   A_21_A700Z1.CmdFaultReset := FALSE;
   A_21_A700Z1.InLocal := FALSE;
   A_21_A700Z1.spare0305 := FALSE;
   A_21_A700Z1.InReport := FALSE;
   A_21_A700Z1.OutTimeoutTime := FALSE;
   A_21_A700Z1.InHWStop := FALSE;
   A_21_A700Z1.InDPFault := FALSE;
   A_21_A700Z1.OutPreAlarmTrue := FALSE;
   A_21_A700Z1.OutPreAlarmFalse := FALSE;
   A_21_A700Z1.OutFlagPos := FALSE;
   A_21_A700Z1.OutFlagNeg := FALSE;
   A_21_A700Z1.OutpFaultReset := FALSE;
   A_21_A700Z1.OutTrue := FALSE;
   A_21_A700Z1.StFalse := FALSE;
   A_21_A700Z1.StCtoTrue := FALSE;
   A_21_A700Z1.StTrue := FALSE;
   A_21_A700Z1.StCtoFalse := FALSE;
   A_21_A700Z1.StFault := FALSE;
   A_21_A700Z1.OutAlarmNrLog := 0;
   A_21_A700Z1.Par.ParObjectNo := 533;
   A_21_A700Z1.Par.ParMsgType := 7147;
   A_21_A700Z1.Par.ParHornCode := 2;
   A_21_A700Z1.Par.ParLogOff := FALSE;
   A_21_A700Z1.Par.spare0401 := FALSE;
   A_21_A700Z1.Par.Par2WorkingCond := FALSE;
   A_21_A700Z1.Par.ParFaultRetry := FALSE;
   A_21_A700Z1.Par.ParBinLevel := FALSE;
   A_21_A700Z1.Par.ParDelayChange := 0;
   A_21_A700Z1.Par.ParDelayTrue := 10;
   A_21_A700Z1.Par.ParDelayFalse := 0;
   A_21_A700Z1.Par.ParTimeoutTrue := 0;
   A_21_A700Z1.Par.ParTimeoutFalse := 0;
   A_21_A700Z1.Par.OutMonTime := 0;
   A_21_A700Z1.Par.OutTransitionTime := 0;
   A_21_A700Z1.Par.OutMonTrue := FALSE;
   A_21_A700Z1.Par.OutMonFalse := FALSE;
   A_21_A700Z1.Par.OutFlagFaultDev := FALSE;
   A_21_A700Z1.Par.OutDelayTime := 0;
   A_21_A800Z1.StCode := 0;
   A_21_A800Z1.InMonTrue := FALSE;
   A_21_A800Z1.InMonFalse := FALSE;
   A_21_A800Z1.InPreAlarmTrue := FALSE;
   A_21_A800Z1.InPreAlarmFalse := FALSE;
   A_21_A800Z1.InStopTrueTime := FALSE;
   A_21_A800Z1.InStopFalseTime := FALSE;
   A_21_A800Z1.InpTrue := FALSE;
   A_21_A800Z1.InpFaultDev := FALSE;
   A_21_A800Z1.CmdRstTrueTime := FALSE;
   A_21_A800Z1.CmdRstFalseTime := FALSE;
   A_21_A800Z1.CmdRunTimeoutTime := FALSE;
   A_21_A800Z1.CmdFaultReset := FALSE;
   A_21_A800Z1.InLocal := FALSE;
   A_21_A800Z1.spare0305 := FALSE;
   A_21_A800Z1.InReport := FALSE;
   A_21_A800Z1.OutTimeoutTime := FALSE;
   A_21_A800Z1.InHWStop := FALSE;
   A_21_A800Z1.InDPFault := FALSE;
   A_21_A800Z1.OutPreAlarmTrue := FALSE;
   A_21_A800Z1.OutPreAlarmFalse := FALSE;
   A_21_A800Z1.OutFlagPos := FALSE;
   A_21_A800Z1.OutFlagNeg := FALSE;
   A_21_A800Z1.OutpFaultReset := FALSE;
   A_21_A800Z1.OutTrue := FALSE;
   A_21_A800Z1.StFalse := FALSE;
   A_21_A800Z1.StCtoTrue := FALSE;
   A_21_A800Z1.StTrue := FALSE;
   A_21_A800Z1.StCtoFalse := FALSE;
   A_21_A800Z1.StFault := FALSE;
   A_21_A800Z1.OutAlarmNrLog := 0;
   A_21_A800Z1.Par.ParObjectNo := 534;
   A_21_A800Z1.Par.ParMsgType := 7147;
   A_21_A800Z1.Par.ParHornCode := 2;
   A_21_A800Z1.Par.ParLogOff := FALSE;
   A_21_A800Z1.Par.spare0401 := FALSE;
   A_21_A800Z1.Par.Par2WorkingCond := FALSE;
   A_21_A800Z1.Par.ParFaultRetry := FALSE;
   A_21_A800Z1.Par.ParBinLevel := FALSE;
   A_21_A800Z1.Par.ParDelayChange := 0;
   A_21_A800Z1.Par.ParDelayTrue := 10;
   A_21_A800Z1.Par.ParDelayFalse := 0;
   A_21_A800Z1.Par.ParTimeoutTrue := 0;
   A_21_A800Z1.Par.ParTimeoutFalse := 0;
   A_21_A800Z1.Par.OutMonTime := 0;
   A_21_A800Z1.Par.OutTransitionTime := 0;
   A_21_A800Z1.Par.OutMonTrue := FALSE;
   A_21_A800Z1.Par.OutMonFalse := FALSE;
   A_21_A800Z1.Par.OutFlagFaultDev := FALSE;
   A_21_A800Z1.Par.OutDelayTime := 0;
      #A_21_A106Z1.Par.ParObjectNo                             :=535;
      #A_21_A106Z1.Par.ParMsgType                              :=7171;
      #A_21_A106Z1.Par.ParHornCode                             :=2;
      #A_21_A106Z1.Par.ParDelayChange                          :=0;
      #A_21_A106Z1.Par.ParDelayTrue                            :=10;
      #A_21_A106Z1.Par.ParDelayFalse                           :=0;
      #A_21_A106Z1.Par.ParTimeoutTrue                          :=0;
      #A_21_A106Z1.Par.ParTimeoutFalse                         :=0;
      #A_21_A106Z1.Par.ParLogOff                               :=False;
      #A_21_A106Z1.Par.Par2WorkingCond                         :=False;
      #A_21_A106Z1.Par.ParFaultRetry                           :=False;
      #A_21_A106Z1.Par.ParBinLevel                             :=False;
END_DATA_BLOCK

